// SIMATIC S7-200 SMART project (STEP 7-Micro/WIN SMART), CPU SR20

SYMBOL_TABLE 主循环
FLUSH_COUNT      VW6020   // 余数
FLUSH_SEL        VW6022   // 商
FMAIN_COUNT_D    VD6010
FMAIN_COUNT_INT  VW6010
IL_COUNT_D       VD6000
IL_COUNT_INT     VW6000
OUTPUT_COUNT_INT VW8000
PUMP_EN          VW6030
TIME_AIR         VW2506
TIME_FLUSH       VW2504
TIME_IL          VW2500
TIME_MESSURE     VW2502
AIL_COUNT        VW2508
CH               VW2510
END_SYMBOL_TABLE

SYMBOL_TABLE 系统符号
Always_On        SM0.0    // 始终接通
END_SYMBOL_TABLE

SYMBOL_TABLE 浓度数据
O2_ZERO          VD4120
O2_R             VD4300
CO_R             VD4304
CO_ZERO          VD336
O2_CALGAS        VD7104   // 标定
CO_CALGAS        VD7100   // 标定
O2_B             VD7004   // 标定
CO_B             VD7000   // 标定
O2_FS            VD320
CO_FS            VD316
CO_NOW           VD108
O2_NOW           VD100
O2_MIT           VD388
CO_MIT           VD376
O2_MIN           VD440
CO_MAX           VD444
END_SYMBOL_TABLE

SYMBOL_TABLE 压力数据
IFP0             VD716
P_0              VD700
P_1              VD704
P_2              VD708
P_3              VD712
END_SYMBOL_TABLE

SYMBOL_TABLE 伴热反吹
TC_0             VD800
BR_T_MIN         VD4132
BR_T_MAX         VD4128
TC_MIN           VD400
P_MIN            VD408
P_MAX            VD412
END_SYMBOL_TABLE

SYMBOL_TABLE 显示
CO0              VD216
CO1              VD220
CO2              VD224
CO3              VD228
O20              VD200
O21              VD204
O22              VD208
O23              VD212
END_SYMBOL_TABLE

SYMBOL_TABLE 中间数据
O2_DI            VD104
O2_HI            VW0
O2_LO            VW2
CO_INT           VW4
TC_HI            VW6
TC_LO            VW8
TC_HI_DI         VD80
TC_LO_DI         VD84
END_SYMBOL_TABLE

SYMBOL_TABLE 串口数据
INT16_0          VW3004
INT16_1          VW3006
INT16_2          VW3008
INT16_3          VW3010
INT16_4          VW3012
END_SYMBOL_TABLE

SYMBOL_TABLE 循环时间
TIME_IL_DEFAULT  VW5000
TIME_MESSURE_DEFAULT VW5002
TIME_FLUSH_DEFAULT VW5004
TIME_AIR_DEFAULT VW5006
END_SYMBOL_TABLE

ORGANIZATION_BLOCK MAIN:OB1
TITLE=气体分析仪程序MAIN
BEGIN
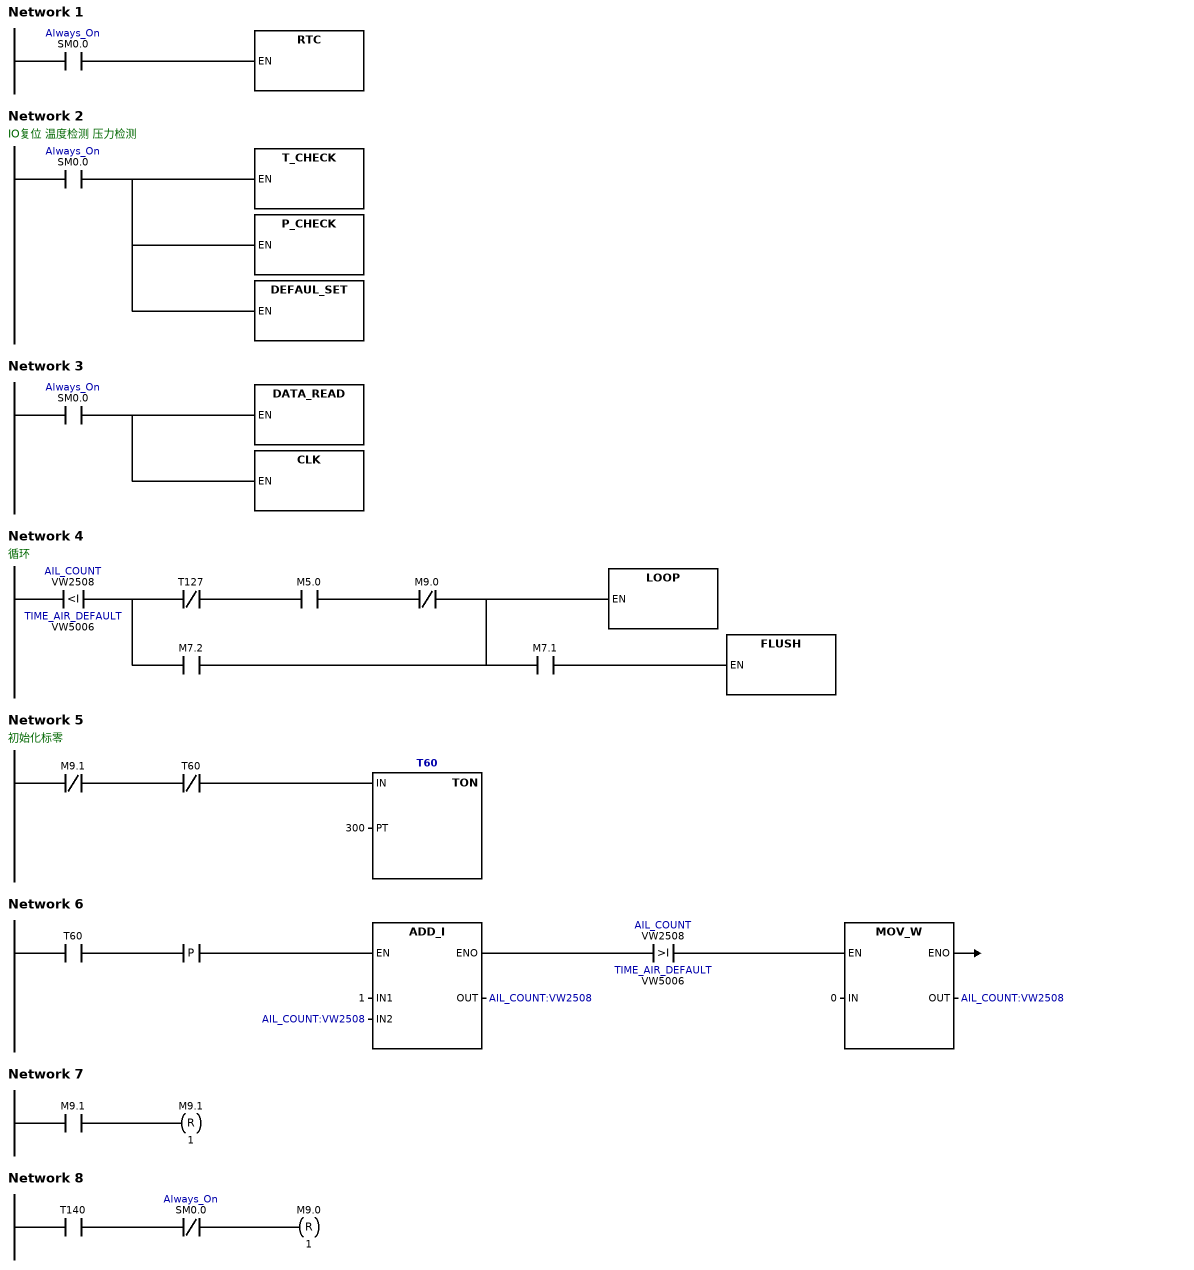
Network 1
LD     Always_On:SM0.0
CALL   RTC:SBR14
Network 2
// IO复位 温度检测 压力检测
LD     Always_On:SM0.0
CALL   T_CHECK:SBR5
CALL   P_CHECK:SBR0
CALL   DEFAUL_SET:SBR20
Network 3
LD     Always_On:SM0.0
CALL   DATA_READ:SBR9
CALL   CLK:SBR19
Network 4
// 循环
LDW<   AIL_COUNT:VW2508, TIME_AIR_DEFAULT:VW5006
LDN    T127
A      M5.0
AN     M9.0
O      M7.2
ALD
CALL   LOOP:SBR6
A      M7.1
CALL   FLUSH:SBR13
Network 5
// 初始化标零
LDN    M9.1
AN     T60
TON    T60, 300
Network 6
LD     T60
EU
+I     1, AIL_COUNT:VW2508
AENO
AW>    AIL_COUNT:VW2508, TIME_AIR_DEFAULT:VW5006
MOVW   0, AIL_COUNT:VW2508
Network 7
LD     M9.1
R      M9.1, 1
Network 8
LD     T140
AN     Always_On:SM0.0
R      M9.0, 1
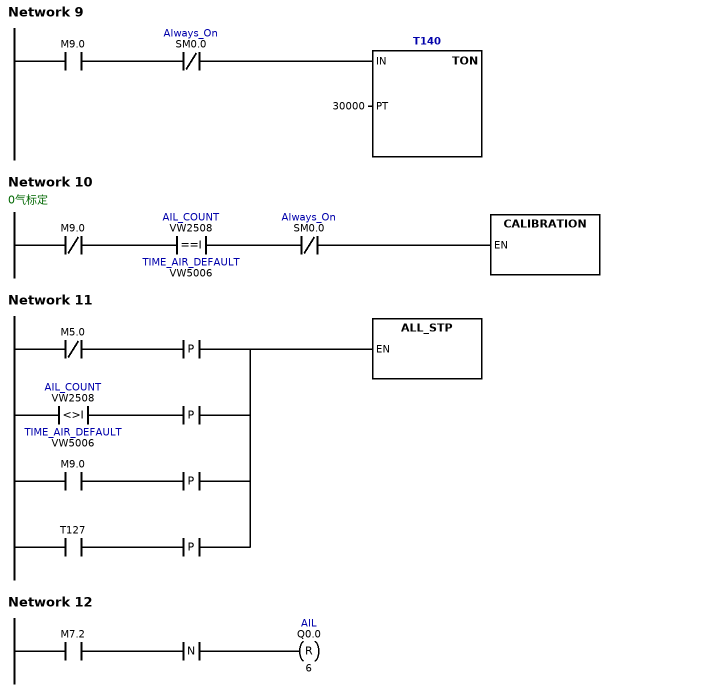
Network 9
LD     M9.0
AN     Always_On:SM0.0
TON    T140, 30000
Network 10
// 0气标定
LDN    M9.0
AW=    AIL_COUNT:VW2508, TIME_AIR_DEFAULT:VW5006
AN     Always_On:SM0.0
CALL   CALIBRATION:SBR4
Network 11
LDN    M5.0
EU
LDW<>  AIL_COUNT:VW2508, TIME_AIR_DEFAULT:VW5006
EU
OLD
LD     M9.0
EU
OLD
LD     T127
EU
OLD
CALL   ALL_STP:SBR15
Network 12
LD     M7.2
ED
R      AIL:Q0.0, 6
END_ORGANIZATION_BLOCK

SUBROUTINE_BLOCK P_CHECK:SBR0
TITLE=反吹压强监测、堵塞监测
BEGIN
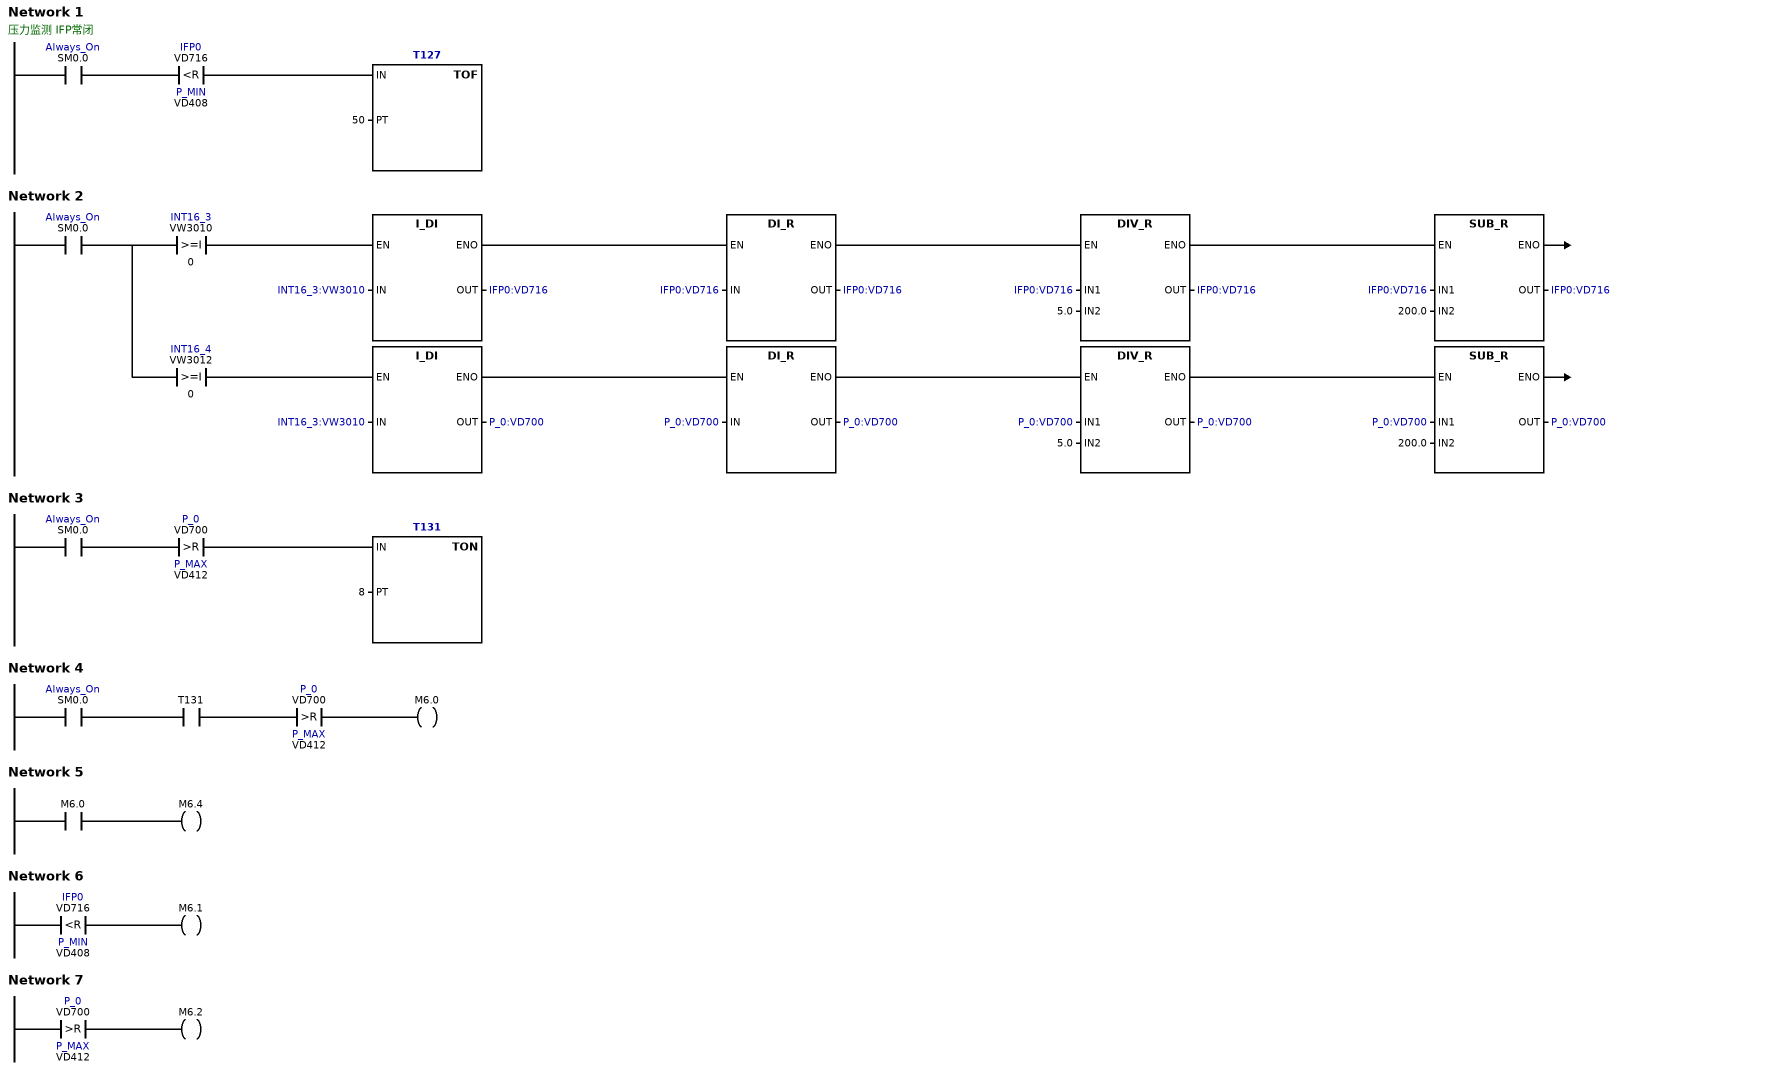
Network 1
// 压力监测 IFP常闭
LD     Always_On:SM0.0
AR<    IFP0:VD716, P_MIN:VD408
TOF    T127, 50
Network 2
LD     Always_On:SM0.0
LPS
AW>=   INT16_3:VW3010, 0
ITD    INT16_3:VW3010, IFP0:VD716
AENO
DTR    IFP0:VD716, IFP0:VD716
AENO
/R     5.0, IFP0:VD716
AENO
-R     200.0, IFP0:VD716
LPP
AW>=   INT16_4:VW3012, 0
ITD    INT16_3:VW3010, P_0:VD700
AENO
DTR    P_0:VD700, P_0:VD700
AENO
/R     5.0, P_0:VD700
AENO
-R     200.0, P_0:VD700
Network 3
LD     Always_On:SM0.0
AR>    P_0:VD700, P_MAX:VD412
TON    T131, 8
Network 4
LD     Always_On:SM0.0
A      T131
AR>    P_0:VD700, P_MAX:VD412
=      M6.0
Network 5
LD     M6.0
=      M6.4
Network 6
LDR<   IFP0:VD716, P_MIN:VD408
=      M6.1
Network 7
LDR>   P_0:VD700, P_MAX:VD412
=      M6.2
END_SUBROUTINE_BLOCK

// SBR1: protected block, not included

// SBR2: protected block, not included

// SBR3: protected block, not included

SUBROUTINE_BLOCK CALIBRATION:SBR4
TITLE=开机空气标定
BEGIN
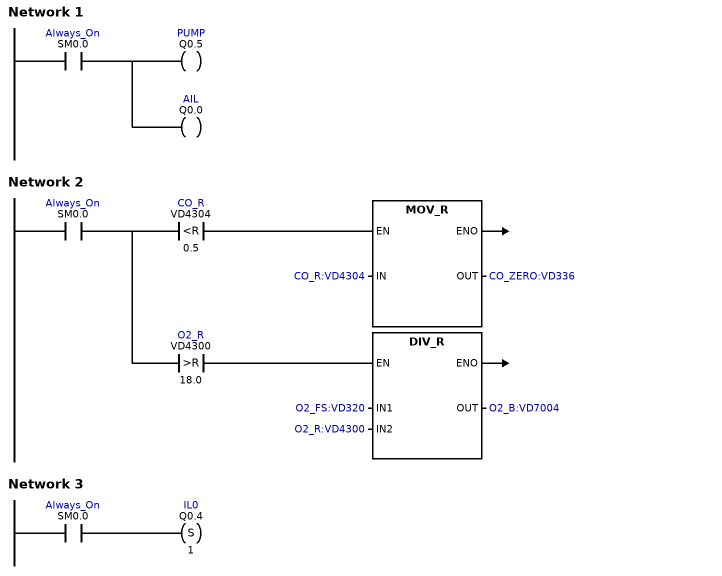
Network 1
LD     Always_On:SM0.0
=      PUMP:Q0.5
=      AIL:Q0.0
Network 2
LD     Always_On:SM0.0
LPS
AR<    CO_R:VD4304, 0.5
MOVR   CO_R:VD4304, CO_ZERO:VD336
LPP
AR>    O2_R:VD4300, 18.0
MOVR   O2_FS:VD320, O2_B:VD7004
/R     O2_R:VD4300, O2_B:VD7004
Network 3
LD     Always_On:SM0.0
S      IL0:Q0.4, 1
END_SUBROUTINE_BLOCK

SUBROUTINE_BLOCK T_CHECK:SBR5
TITLE=冷凝器温度、炉膛壁温度监测
BEGIN
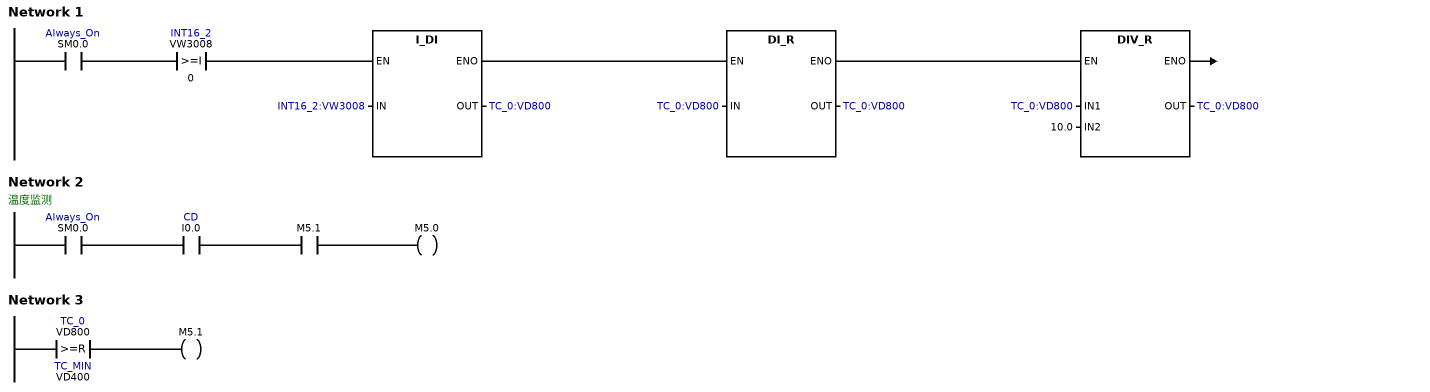
Network 1
LD     Always_On:SM0.0
AW>=   INT16_2:VW3008, 0
ITD    INT16_2:VW3008, TC_0:VD800
AENO
DTR    TC_0:VD800, TC_0:VD800
AENO
/R     10.0, TC_0:VD800
Network 2
// 温度监测
LD     Always_On:SM0.0
A      CD:I0.0
A      M5.1
=      M5.0
Network 3
LDR>=  TC_0:VD800, TC_MIN:VD400
=      M5.1
END_SUBROUTINE_BLOCK

SUBROUTINE_BLOCK LOOP:SBR6
TITLE=子程序注释
BEGIN
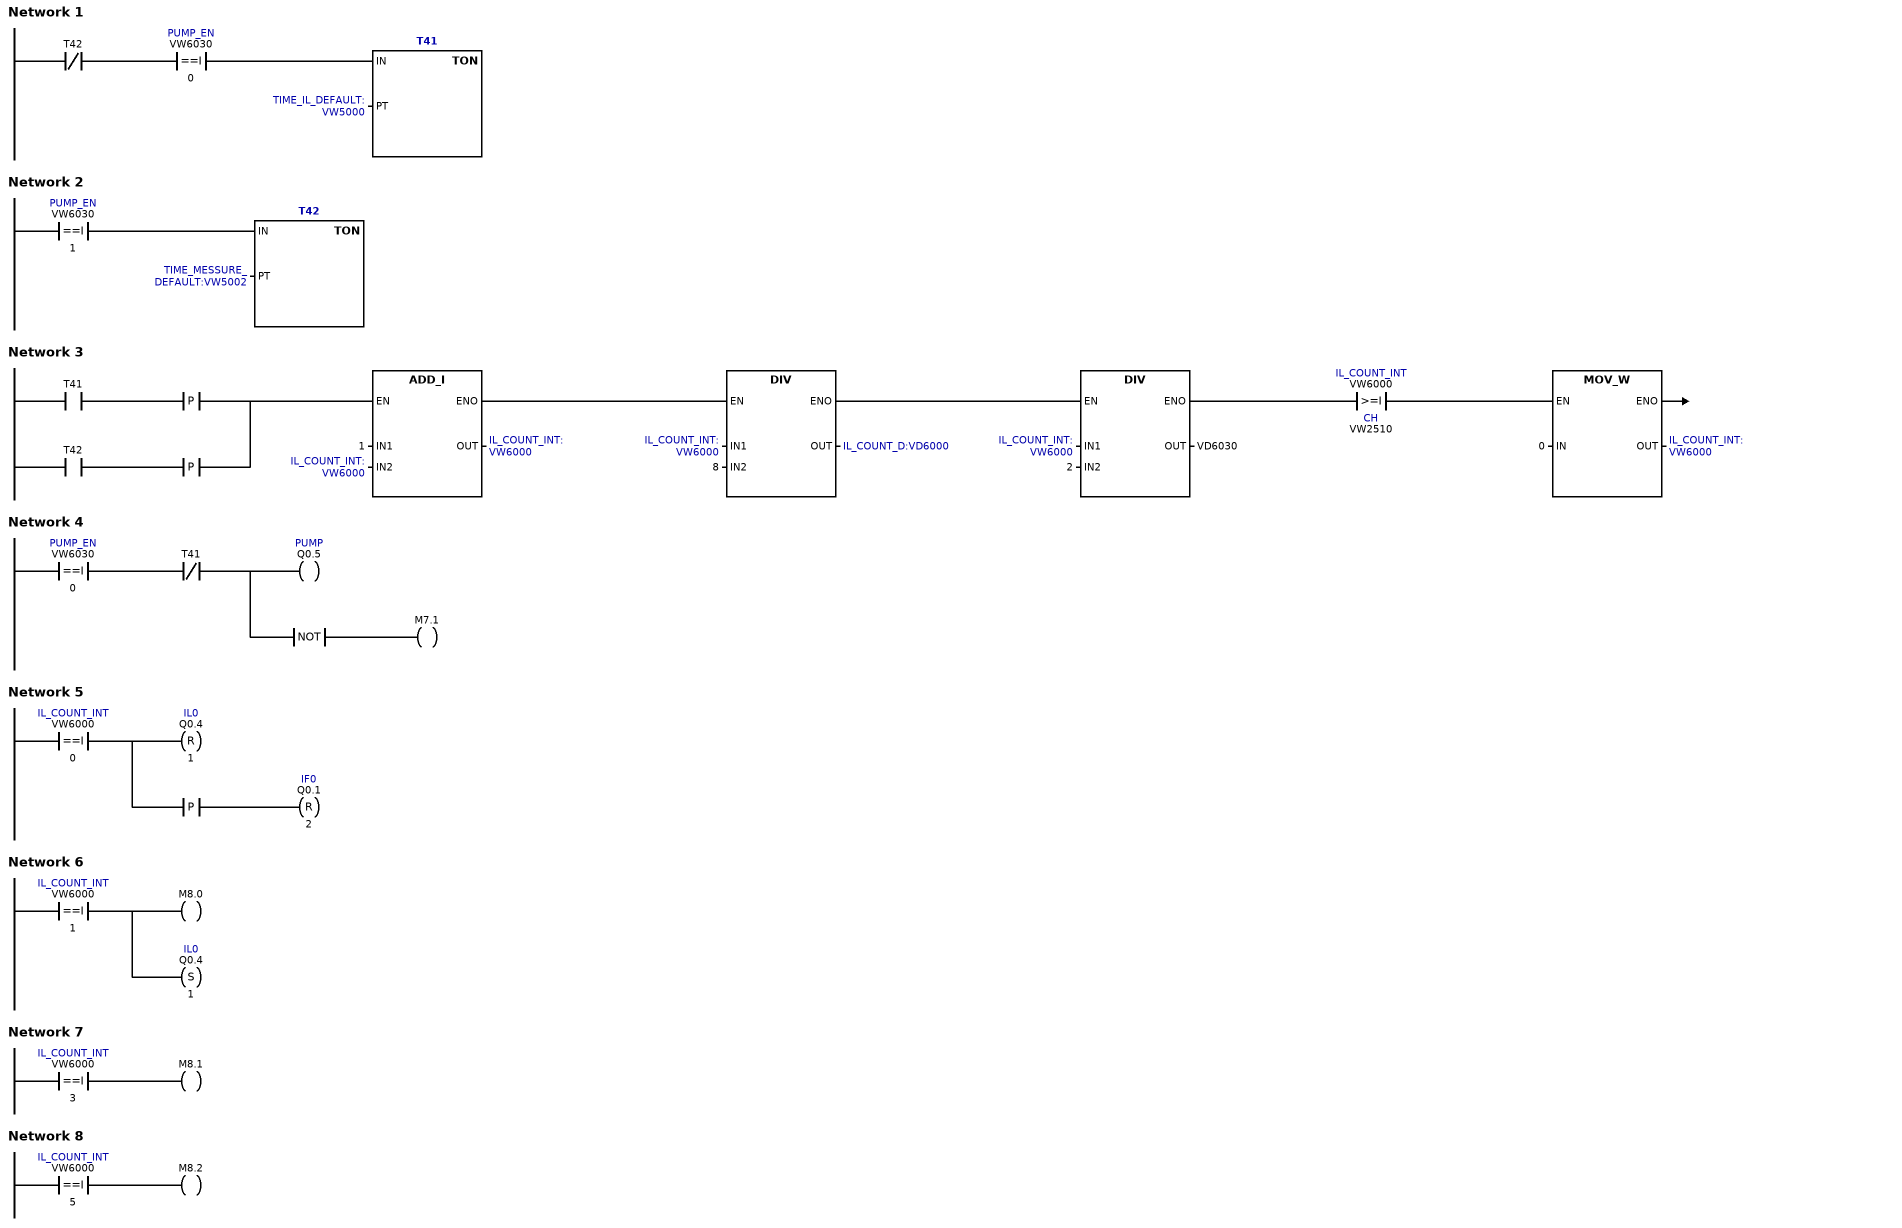
Network 1
LDN    T42
AW=    PUMP_EN:VW6030, 0
TON    T41, TIME_IL_DEFAULT:VW5000
Network 2
LDW=   PUMP_EN:VW6030, 1
TON    T42, TIME_MESSURE_DEFAULT:VW5002
Network 3
LD     T41
EU
LD     T42
EU
OLD
+I     1, IL_COUNT_INT:VW6000
AENO
MOVW   IL_COUNT_INT:VW6000, VW6002
AENO
DIV    8, IL_COUNT_D:VD6000
AENO
MOVW   IL_COUNT_INT:VW6000, VW6032
AENO
DIV    2, VD6030
AENO
AW>=   IL_COUNT_INT:VW6000, CH:VW2510
MOVW   0, IL_COUNT_INT:VW6000
Network 4
LDW=   PUMP_EN:VW6030, 0
AN     T41
=      PUMP:Q0.5
NOT
=      M7.1
Network 5
LDW=   IL_COUNT_INT:VW6000, 0
R      IL0:Q0.4, 1
EU
R      IF0:Q0.1, 2
Network 6
LDW=   IL_COUNT_INT:VW6000, 1
=      M8.0
S      IL0:Q0.4, 1
Network 7
LDW=   IL_COUNT_INT:VW6000, 3
=      M8.1
Network 8
LDW=   IL_COUNT_INT:VW6000, 5
=      M8.2
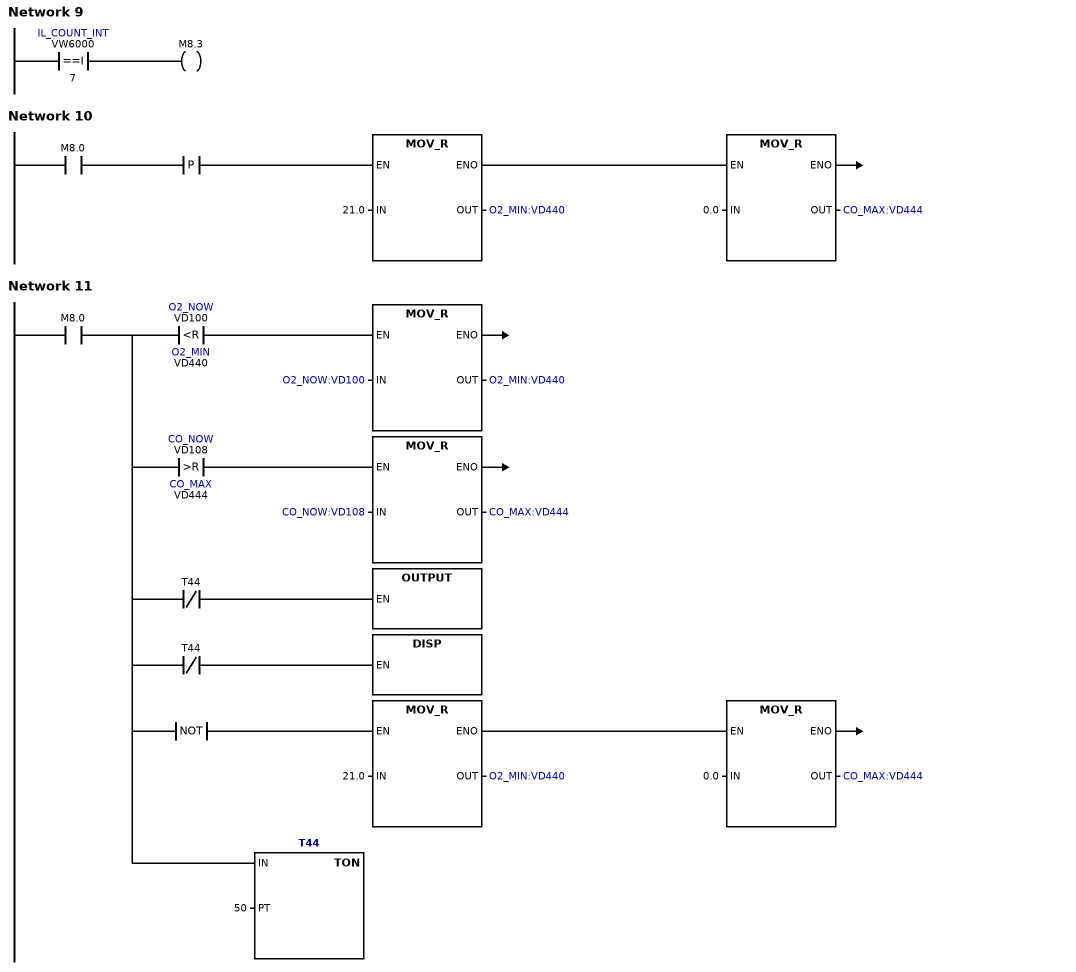
Network 9
LDW=   IL_COUNT_INT:VW6000, 7
=      M8.3
Network 10
LD     M8.0
EU
MOVR   21.0, O2_MIN:VD440
AENO
MOVR   0.0, CO_MAX:VD444
Network 11
LD     M8.0
LPS
AR<    O2_NOW:VD100, O2_MIN:VD440
MOVR   O2_NOW:VD100, O2_MIN:VD440
LRD
AR>    CO_NOW:VD108, CO_MAX:VD444
MOVR   CO_NOW:VD108, CO_MAX:VD444
LRD
AN     T44
CALL   OUTPUT:SBR8
LRD
AN     T44
CALL   DISP:SBR18
LRD
NOT
MOVR   21.0, O2_MIN:VD440
AENO
MOVR   0.0, CO_MAX:VD444
LPP
TON    T44, 50
END_SUBROUTINE_BLOCK

SUBROUTINE_BLOCK OUTPUT:SBR8
TITLE=写输出模块
BEGIN
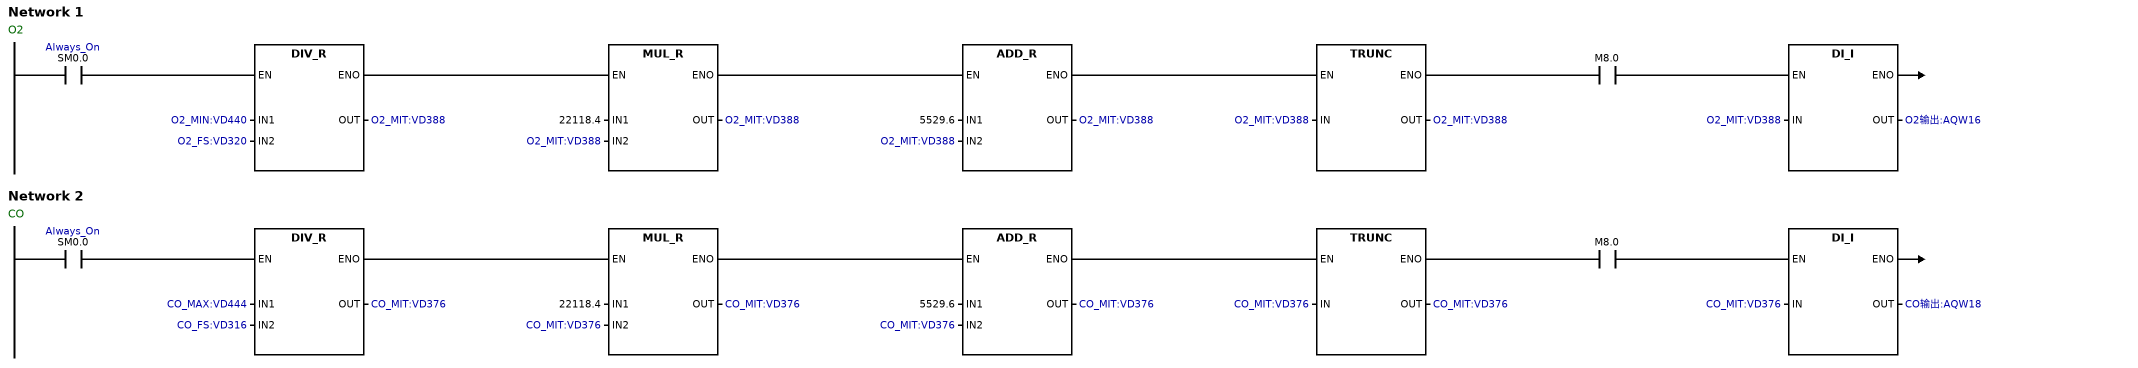
Network 1
// O2
LD     Always_On:SM0.0
MOVR   O2_MIN:VD440, O2_MIT:VD388
AENO
/R     O2_FS:VD320, O2_MIT:VD388
AENO
*R     22118.4, O2_MIT:VD388
AENO
+R     5529.6, O2_MIT:VD388
AENO
TRUNC  O2_MIT:VD388, O2_MIT:VD388
AENO
A      M8.0
DTI    O2_MIT:VD388, O2输出:AQW16
Network 2
// CO
LD     Always_On:SM0.0
MOVR   CO_MAX:VD444, CO_MIT:VD376
AENO
/R     CO_FS:VD316, CO_MIT:VD376
AENO
*R     22118.4, CO_MIT:VD376
AENO
+R     5529.6, CO_MIT:VD376
AENO
TRUNC  CO_MIT:VD376, CO_MIT:VD376
AENO
A      M8.0
DTI    CO_MIT:VD376, CO输出:AQW18
END_SUBROUTINE_BLOCK

SUBROUTINE_BLOCK DATA_READ:SBR9
TITLE=读参数
BEGIN
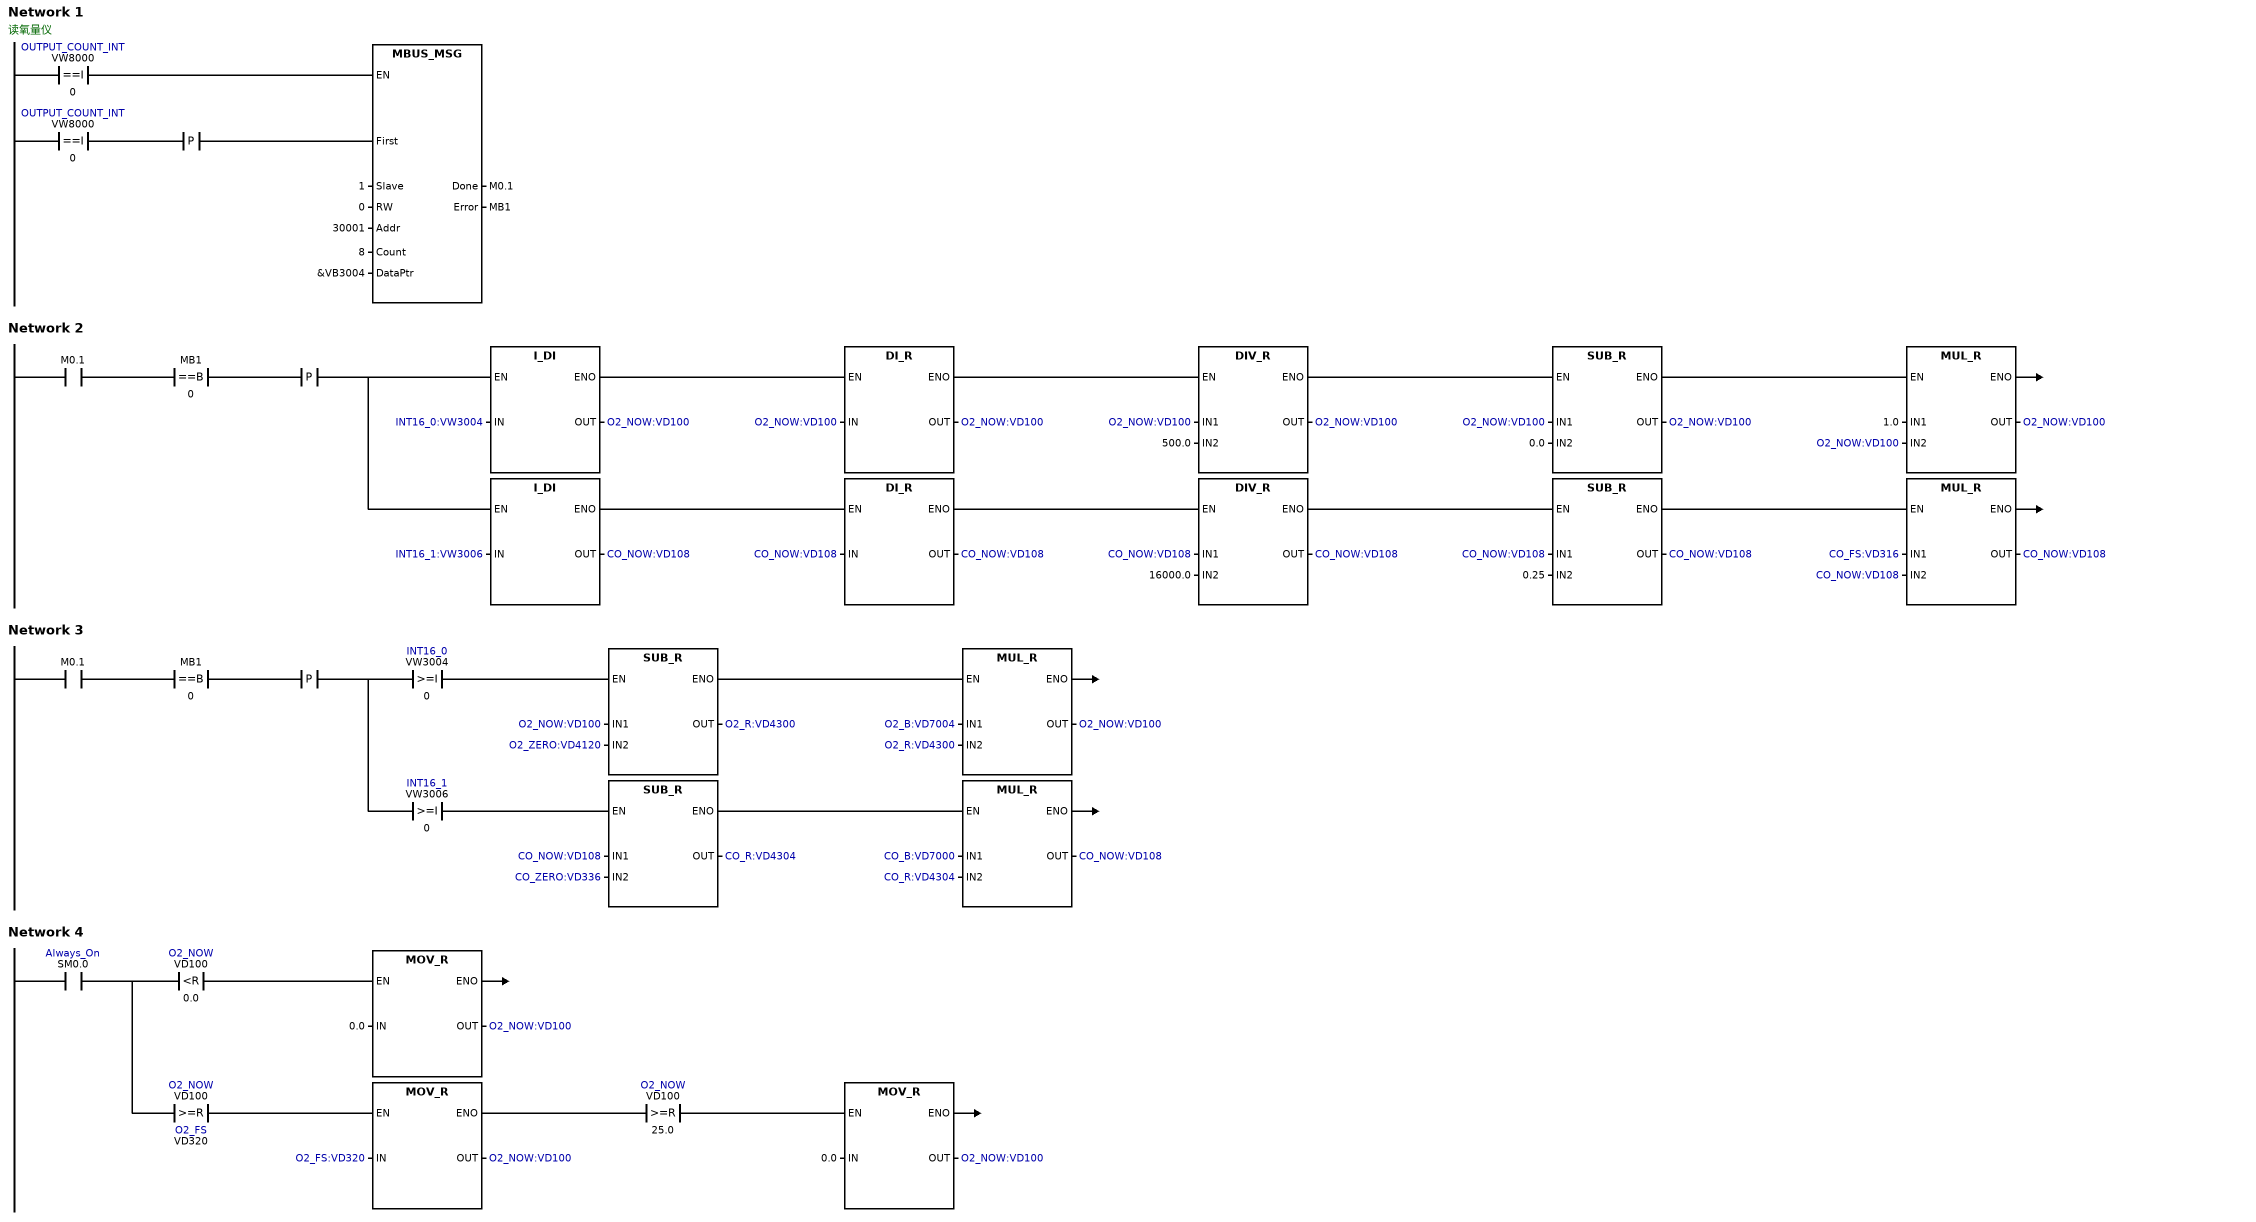
Network 1
// 读氧量仪
LDW=   OUTPUT_COUNT_INT:VW8000, 0
=      L60.0
LDW=   OUTPUT_COUNT_INT:VW8000, 0
EU
=      L63.7
LD     L60.0
CALL   MBUS_MSG:SBR2, L63.7, 1, 0, 30001, 8, &VB3004, M0.1, MB1
Network 2
LD     M0.1
AB=    MB1, 0
EU
LPS
ITD    INT16_0:VW3004, O2_NOW:VD100
AENO
DTR    O2_NOW:VD100, O2_NOW:VD100
AENO
/R     500.0, O2_NOW:VD100
AENO
-R     0.0, O2_NOW:VD100
AENO
*R     1.0, O2_NOW:VD100
LPP
ITD    INT16_1:VW3006, CO_NOW:VD108
AENO
DTR    CO_NOW:VD108, CO_NOW:VD108
AENO
/R     16000.0, CO_NOW:VD108
AENO
-R     0.25, CO_NOW:VD108
AENO
*R     CO_FS:VD316, CO_NOW:VD108
Network 3
LD     M0.1
AB=    MB1, 0
EU
LPS
AW>=   INT16_0:VW3004, 0
MOVR   O2_NOW:VD100, O2_R:VD4300
AENO
-R     O2_ZERO:VD4120, O2_R:VD4300
AENO
MOVR   O2_B:VD7004, O2_NOW:VD100
*R     O2_R:VD4300, O2_NOW:VD100
LPP
AW>=   INT16_1:VW3006, 0
MOVR   CO_NOW:VD108, CO_R:VD4304
AENO
-R     CO_ZERO:VD336, CO_R:VD4304
AENO
MOVR   CO_B:VD7000, CO_NOW:VD108
*R     CO_R:VD4304, CO_NOW:VD108
Network 4
LD     Always_On:SM0.0
LPS
AR<    O2_NOW:VD100, 0.0
MOVR   0.0, O2_NOW:VD100
LPP
AR>=   O2_NOW:VD100, O2_FS:VD320
MOVR   O2_FS:VD320, O2_NOW:VD100
AENO
AR>=   O2_NOW:VD100, 25.0
MOVR   0.0, O2_NOW:VD100
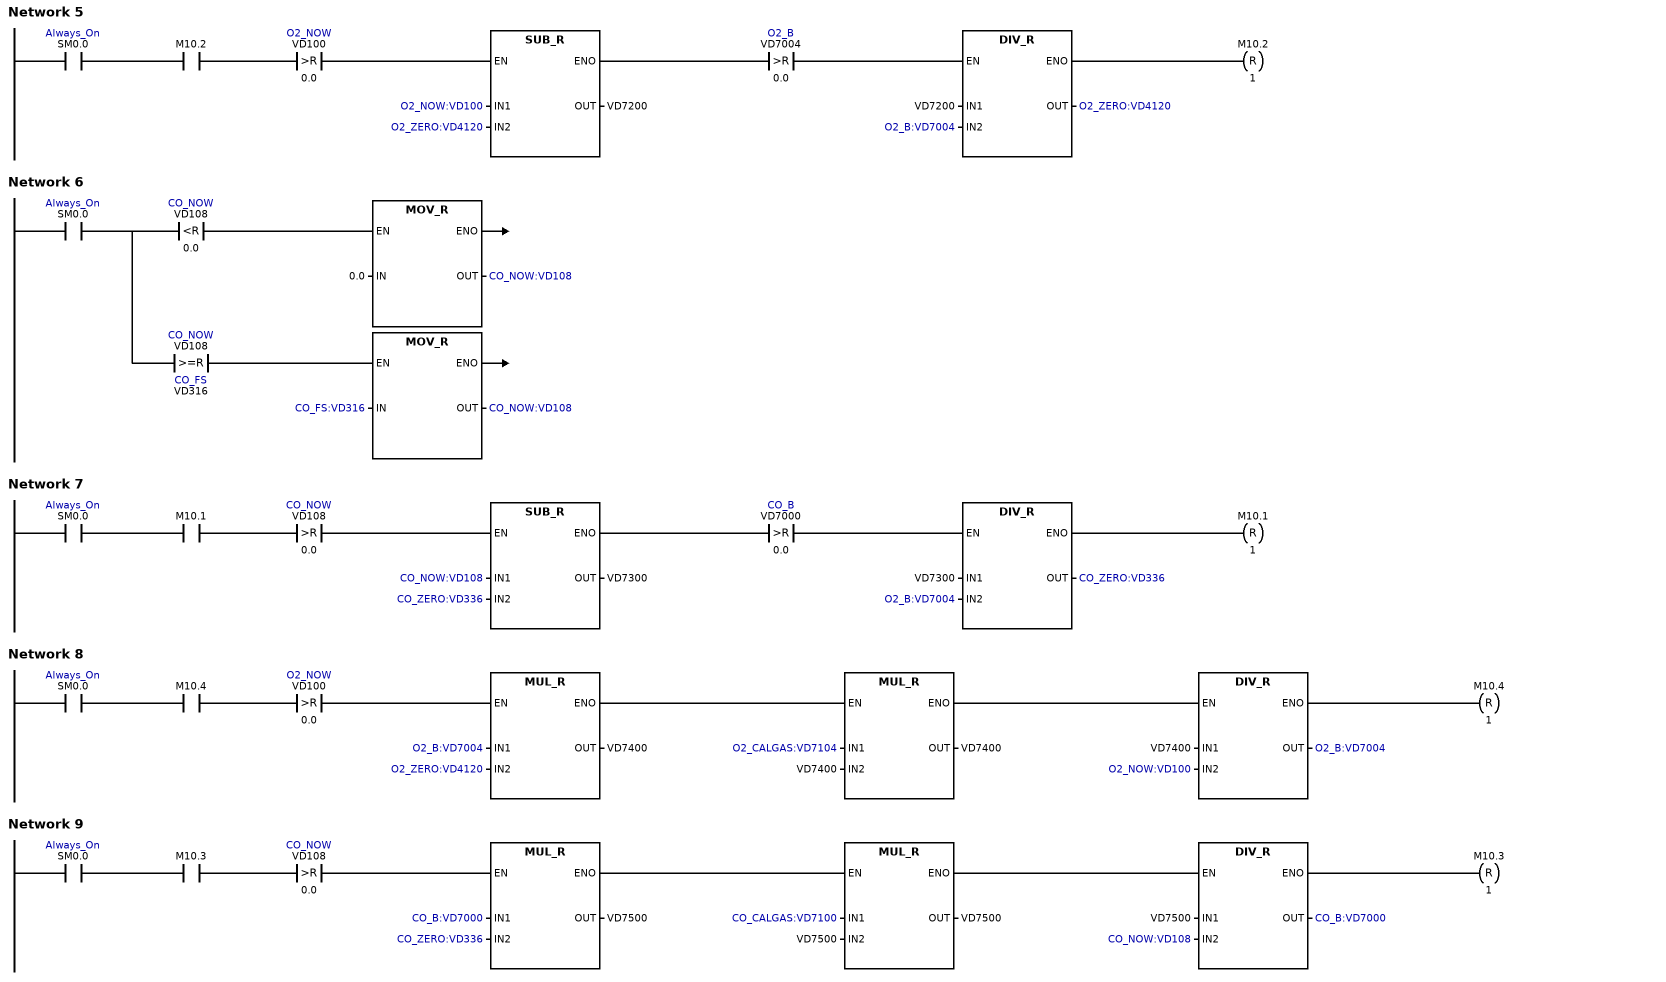
Network 5
LD     Always_On:SM0.0
A      M10.2
AR>    O2_NOW:VD100, 0.0
MOVR   O2_NOW:VD100, VD7200
AENO
-R     O2_ZERO:VD4120, VD7200
AENO
AR>    O2_B:VD7004, 0.0
MOVR   VD7200, O2_ZERO:VD4120
AENO
/R     O2_B:VD7004, O2_ZERO:VD4120
AENO
R      M10.2, 1
Network 6
LD     Always_On:SM0.0
LPS
AR<    CO_NOW:VD108, 0.0
MOVR   0.0, CO_NOW:VD108
LPP
AR>=   CO_NOW:VD108, CO_FS:VD316
MOVR   CO_FS:VD316, CO_NOW:VD108
Network 7
LD     Always_On:SM0.0
A      M10.1
AR>    CO_NOW:VD108, 0.0
MOVR   CO_NOW:VD108, VD7300
AENO
-R     CO_ZERO:VD336, VD7300
AENO
AR>    CO_B:VD7000, 0.0
MOVR   VD7300, CO_ZERO:VD336
AENO
/R     O2_B:VD7004, CO_ZERO:VD336
AENO
R      M10.1, 1
Network 8
LD     Always_On:SM0.0
A      M10.4
AR>    O2_NOW:VD100, 0.0
MOVR   O2_B:VD7004, VD7400
AENO
*R     O2_ZERO:VD4120, VD7400
AENO
*R     O2_CALGAS:VD7104, VD7400
AENO
MOVR   VD7400, O2_B:VD7004
AENO
/R     O2_NOW:VD100, O2_B:VD7004
AENO
R      M10.4, 1
Network 9
LD     Always_On:SM0.0
A      M10.3
AR>    CO_NOW:VD108, 0.0
MOVR   CO_B:VD7000, VD7500
AENO
*R     CO_ZERO:VD336, VD7500
AENO
*R     CO_CALGAS:VD7100, VD7500
AENO
MOVR   VD7500, CO_B:VD7000
AENO
/R     CO_NOW:VD108, CO_B:VD7000
AENO
R      M10.3, 1
END_SUBROUTINE_BLOCK

// SBR10: protected block, not included

// SBR11: protected block, not included

// SBR12: protected block, not included

SUBROUTINE_BLOCK FLUSH:SBR13
TITLE=子程序注释
BEGIN
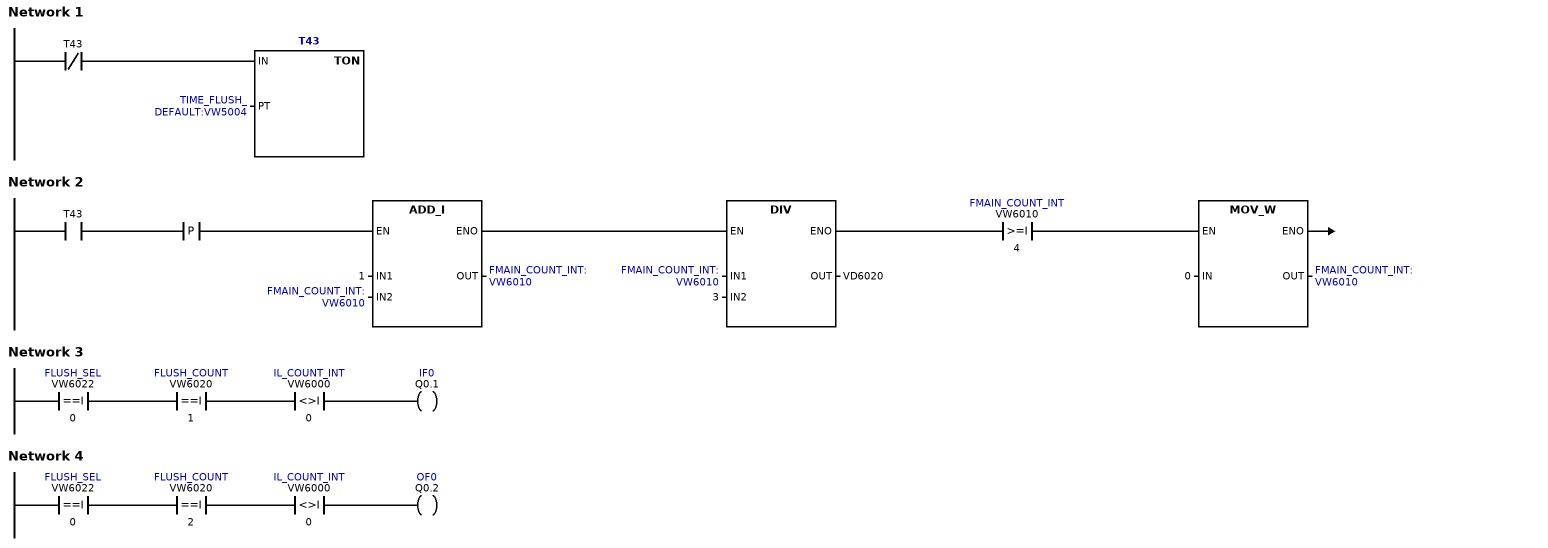
Network 1
LDN    T43
TON    T43, TIME_FLUSH_DEFAULT:VW5004
Network 2
LD     T43
EU
+I     1, FMAIN_COUNT_INT:VW6010
AENO
MOVW   FMAIN_COUNT_INT:VW6010, FLUSH_SEL:VW6022
AENO
DIV    3, VD6020
AENO
AW>=   FMAIN_COUNT_INT:VW6010, 4
MOVW   0, FMAIN_COUNT_INT:VW6010
Network 3
LDW=   FLUSH_SEL:VW6022, 0
AW=    FLUSH_COUNT:VW6020, 1
AW<>   IL_COUNT_INT:VW6000, 0
=      IF0:Q0.1
Network 4
LDW=   FLUSH_SEL:VW6022, 0
AW=    FLUSH_COUNT:VW6020, 2
AW<>   IL_COUNT_INT:VW6000, 0
=      OF0:Q0.2
END_SUBROUTINE_BLOCK

SUBROUTINE_BLOCK RTC:SBR14
TITLE=子程序注释
BEGIN
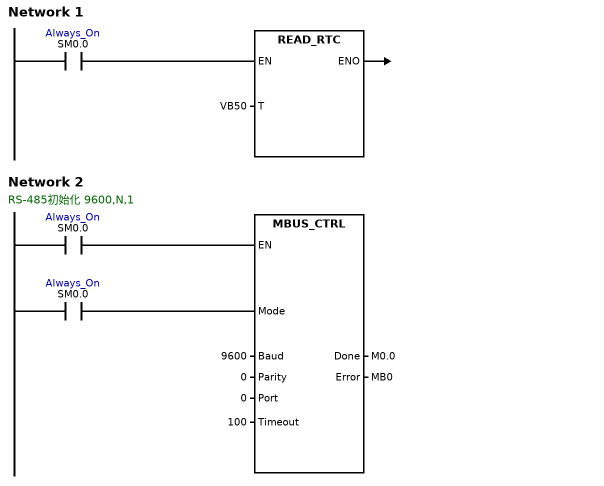
Network 1
LD     Always_On:SM0.0
TODR   VB50
Network 2
// RS-485初始化 9600,N,1
LD     Always_On:SM0.0
=      L60.0
LD     Always_On:SM0.0
=      L63.7
LD     L60.0
CALL   MBUS_CTRL:SBR1, L63.7, 9600, 0, 0, 100, M0.0, MB0
Network 3
// 程序段注释
END_SUBROUTINE_BLOCK

SUBROUTINE_BLOCK ALL_STP:SBR15
TITLE=全部停止
BEGIN
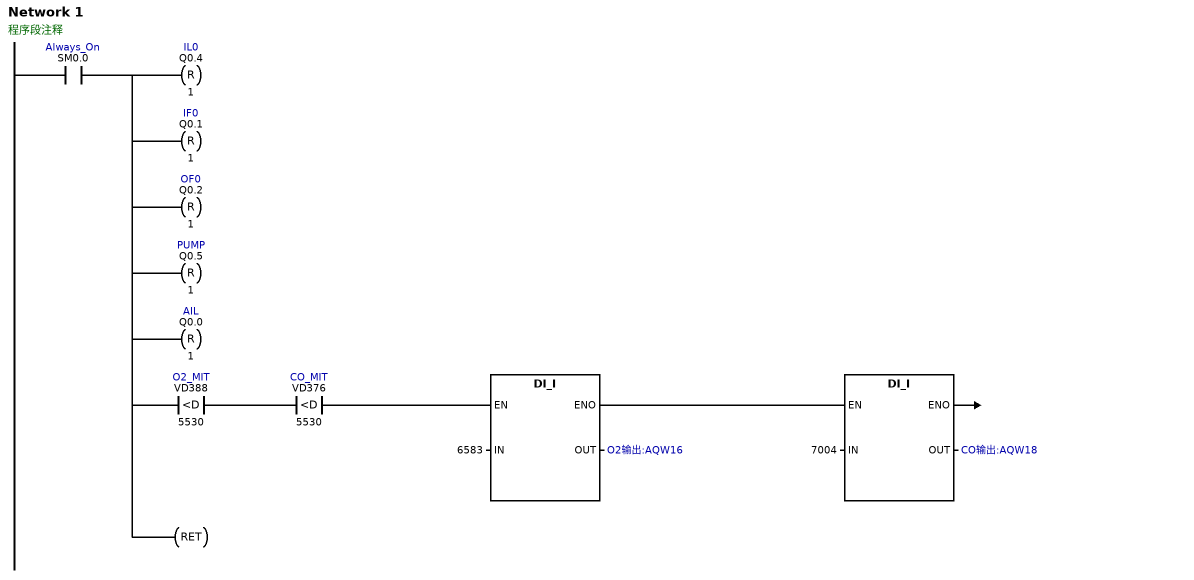
Network 1
// 程序段注释
LD     Always_On:SM0.0
LPS
R      IL0:Q0.4, 1
R      IF0:Q0.1, 1
R      OF0:Q0.2, 1
R      PUMP:Q0.5, 1
R      AIL:Q0.0, 1
AD<    O2_MIT:VD388, 5530
AD<    CO_MIT:VD376, 5530
DTI    6583, O2输出:AQW16
AENO
DTI    7004, CO输出:AQW18
LPP
CRET
END_SUBROUTINE_BLOCK

SUBROUTINE_BLOCK TRAP:SBR16
TITLE=堵塞强制反吹
BEGIN
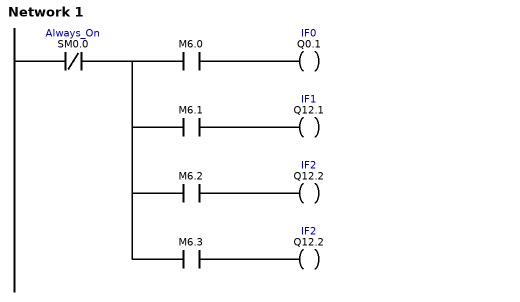
Network 1
LDN    Always_On:SM0.0
LPS
A      M6.0
=      IF0:Q0.1
LRD
A      M6.1
=      IF1:Q12.1
LRD
A      M6.2
=      IF2:Q12.2
LPP
A      M6.3
=      IF2:Q12.2
END_SUBROUTINE_BLOCK

SUBROUTINE_BLOCK CO_READ:SBR17
TITLE=
BEGIN
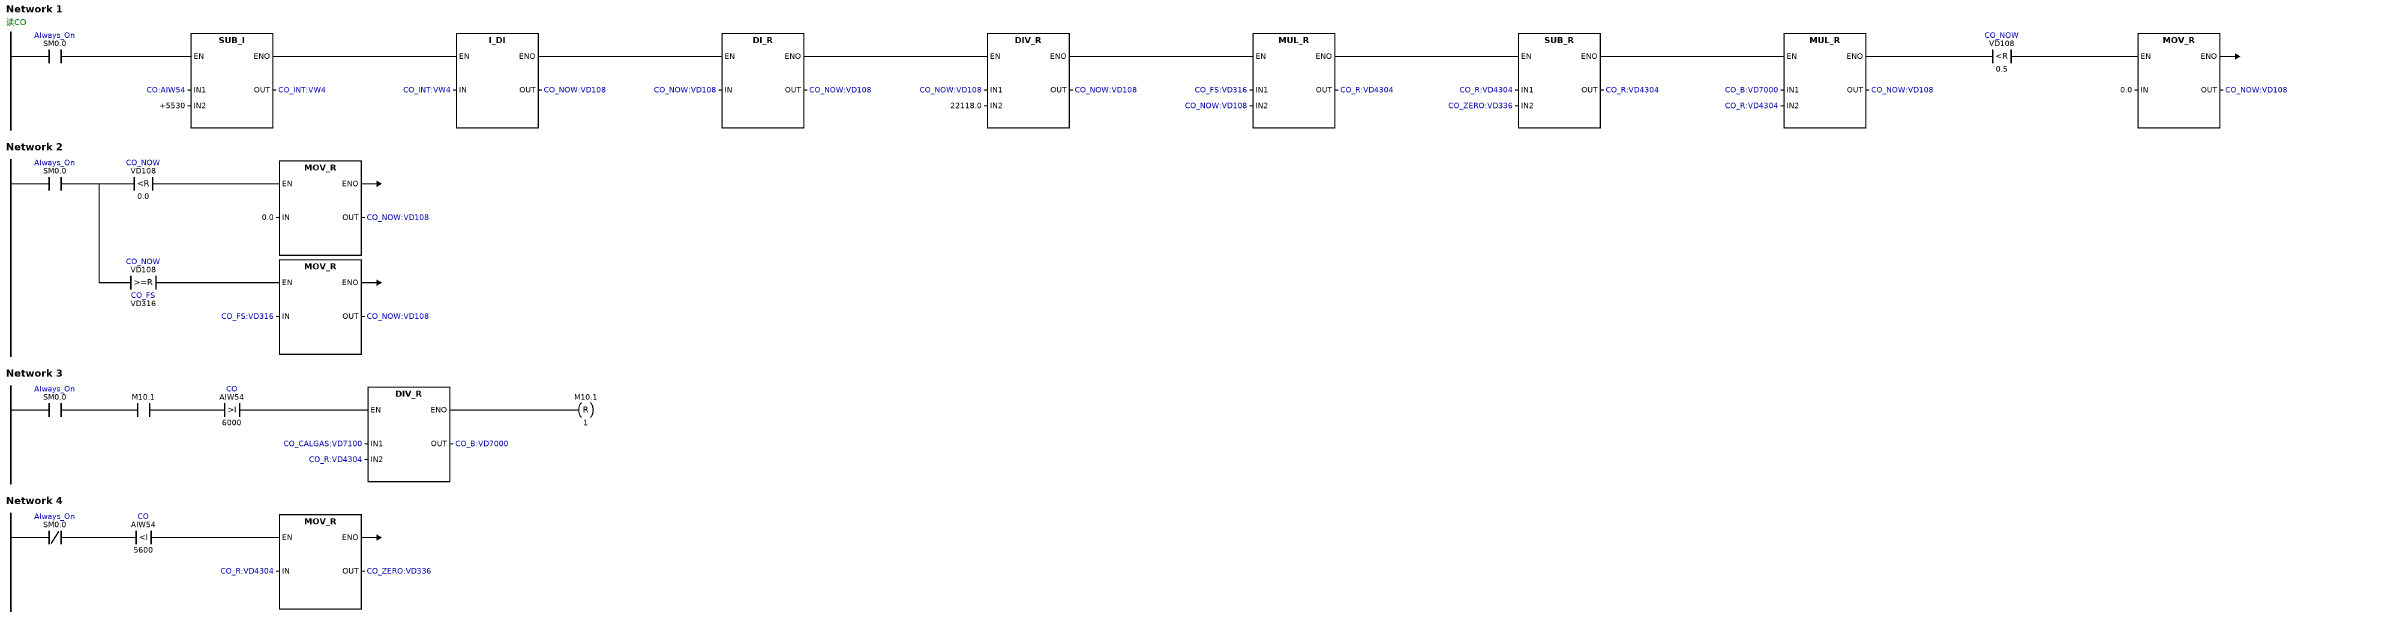
Network 1
// 读CO
LD     Always_On:SM0.0
MOVW   CO:AIW54, CO_INT:VW4
AENO
-I     +5530, CO_INT:VW4
AENO
ITD    CO_INT:VW4, CO_NOW:VD108
AENO
DTR    CO_NOW:VD108, CO_NOW:VD108
AENO
/R     22118.0, CO_NOW:VD108
AENO
MOVR   CO_FS:VD316, CO_R:VD4304
AENO
*R     CO_NOW:VD108, CO_R:VD4304
AENO
-R     CO_ZERO:VD336, CO_R:VD4304
AENO
MOVR   CO_B:VD7000, CO_NOW:VD108
AENO
*R     CO_R:VD4304, CO_NOW:VD108
AENO
AR<    CO_NOW:VD108, 0.5
MOVR   0.0, CO_NOW:VD108
Network 2
LD     Always_On:SM0.0
LPS
AR<    CO_NOW:VD108, 0.0
MOVR   0.0, CO_NOW:VD108
LPP
AR>=   CO_NOW:VD108, CO_FS:VD316
MOVR   CO_FS:VD316, CO_NOW:VD108
Network 3
LD     Always_On:SM0.0
A      M10.1
AW>    CO:AIW54, 6000
MOVR   CO_CALGAS:VD7100, CO_B:VD7000
AENO
/R     CO_R:VD4304, CO_B:VD7000
AENO
R      M10.1, 1
Network 4
LDN    Always_On:SM0.0
AW<    CO:AIW54, 5600
MOVR   CO_R:VD4304, CO_ZERO:VD336
END_SUBROUTINE_BLOCK

SUBROUTINE_BLOCK DISP:SBR18
TITLE=子程序注释
BEGIN
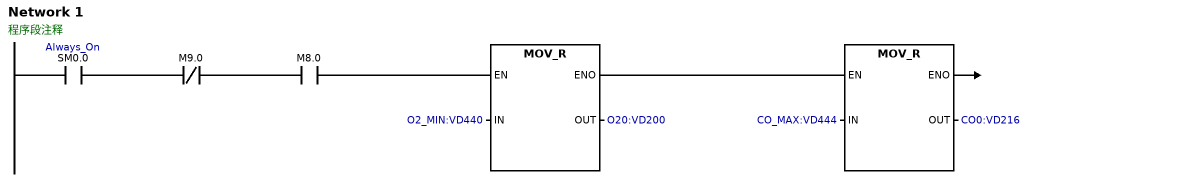
Network 1
// 程序段注释
LD     Always_On:SM0.0
AN     M9.0
A      M8.0
MOVR   O2_MIN:VD440, O20:VD200
AENO
MOVR   CO_MAX:VD444, CO0:VD216
END_SUBROUTINE_BLOCK

DATA_BLOCK_TAB 页面_1
BEGIN
//数据页注释
//阈值
         TC_MIN, 50.0        //TC温度阈值
         BR_T_MIN, 50.0      //伴热温度MIN
         BR_T_MAX, 110.0     //伴热温度MAX
         P_MIN, 10.0         //反吹压强MIN
         P_MAX, 600.0        //反吹压强MAX堵塞
//量程
         CO_FS, 30.0
         O2_FS, 21.0
//计数器初始化
         IL_COUNT_INT, 0
         FMAIN_COUNT_INT, 0
//标定数据default
         O2_CALGAS, 0.0
         CO_CALGAS, 0.0
         O2_ZERO, 0.0        //O2零点
         CO_ZERO, 0.0        //CO零点
         O2_B, 1.0
         CO_B, 1.0
//循环时间
         TIME_IL, 80
         TIME_MESSURE, 16
         TIME_FLUSH, 2
         TIME_AIR, 24
         CH, 2
END_DATA_BLOCK_TAB
